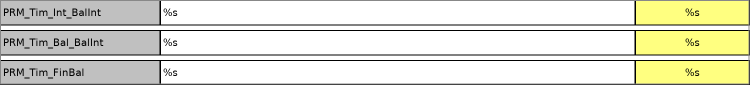
VISUALIZATION VISU_CONFIG_INTERJOINT  // 750x85
(*visualistion pour secondaire dans chambre et primaire dans sas ==> paramètres pour chambre*)
VAR_IN_OUT
	m_Input_Pompage : BLOCK_POMP_1E_PCR_PPM_ASS_ETHERCAT_SINGER;
END_VAR
    Rectangle (160,0 475x25), "%s", text list: 'TextList_Config_Pompage', text index: 17
    Rectangle (635,0 115x25), "%s", text variable: m_Input_Pompage.PRM_Tim_Int_BalInt, input disabled if: NOT Global_Variables.PRG_USER.ACTU_USER.CONF_MACHINE
        OnMouseClick: write the text variable via InputWithLimits
    Rectangle (0,0 160x25), "PRM_Tim_Int_BalInt"
    Rectangle (160,30 475x25), "%s", text list: 'TextList_Config_Pompage', text index: 18
    Rectangle (635,30 115x25), "%s", text variable: m_Input_Pompage.PRM_Tim_Bal_BalInt, input disabled if: NOT Global_Variables.PRG_USER.ACTU_USER.CONF_MACHINE
        OnMouseClick: write the text variable via InputWithLimits
    Rectangle (0,30 160x25), "PRM_Tim_Bal_BalInt"
    Rectangle (0,60 160x25), "PRM_Tim_FinBal"
    Rectangle (160,60 475x25), "%s", text list: 'TextList_Config_Pompage', text index: 19
    Rectangle (635,60 115x25), "%s", text variable: m_Input_Pompage.PRM_Tim_FinBal, input disabled if: NOT Global_Variables.PRG_USER.ACTU_USER.CONF_MACHINE
        OnMouseClick: write the text variable via InputWithLimits
END_VISUALIZATION

// ---- Visualizations/Symbole/POMPES/CRYO_CTI_V4/VISU_ETAPE_REGEN.TcVIS
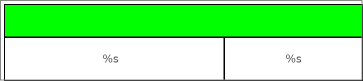
VISUALIZATION VISU_ETAPE_REGEN  // 363x81
VAR_IN_OUT
	COM: BLOCK_RS232_ONBOARD_V4;
END_VAR
    Textfield (4,37 220x44), "%s", text list: 'TextList_CryoPump', text index: COM.STEP_REGEN_ID
    Rectangle (4,4 359x33), colour toggle: COM.STATE_Regen, text list: 'TextList_CryoPump', text index: 43
    Textfield (224,37 139x44), "%s", text variable: COM.VAR_Affichage, text list: 'TextList_CryoPump', text index: COM.ID_ERREUR_REGEN
    Rectangle (4,4 359x33), colour toggle: COM.STATE_Regen, invisible if: not(COM.Regen_completed), text list: 'TextList_CryoPump', text index: 43
END_VISUALIZATION

// ---- Visualizations/Symbole/POMPES/CRYO_CTI_V4/VISU_INFO.TcVIS
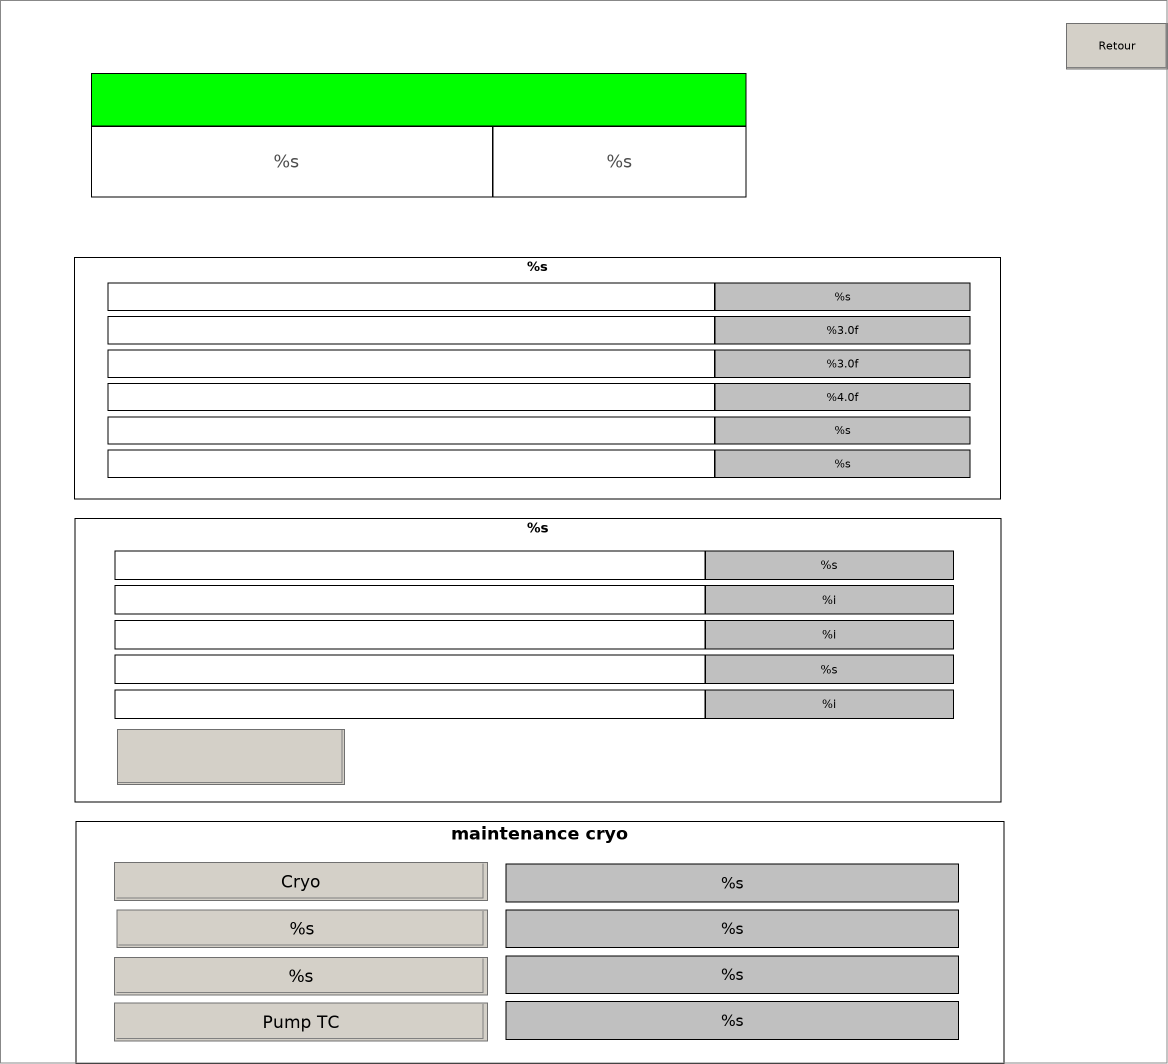
VISUALIZATION VISU_INFO  // 1168x1064
VAR_IN_OUT
	m_Input_CRYO: BLOCK_RS232_ONBOARD_V4;
	m_Input_PRG_POMPAGE: BLOCK_PRG_POMPAGE;
END_VAR
    Button (1066,23 102x46), "Retour", text list: 'GlabalTextList', text index: 16
        OnMouseClick: change screen: Previous SYN_POMPAGE
        OnMouseClick: execute { .VISU_INDEX_MANU := 0; }
    Frame (60,812 944x252), invisible if: NOT Global_Variables.PRG_USER.MANUFACTURER, input disabled if: NOT Global_Variables.PRG_USER.ACTU_USER.CONF_MACHINE OR NOT Global_Variables.PRG_USER.MANUFACTURER
        shows VISU_MAINT_CRYO_AC(COM := m_Input_CRYO)
    Frame (65,509 936x293)
        shows VISU_INFO_SUPP_POMPE(COM := m_Input_CRYO)
    Frame (68,255 933x244)
        shows VISU_RECUPERATION_ETATS(COM := m_Input_CRYO)
    Frame (84,67 662x130)
        shows VISU_ETAPE_REGEN(COM := m_Input_CRYO)
END_VISUALIZATION

// ---- Visualizations/Symbole/POMPES/CRYO_CTI_V4/VISU_INFO_SUPP_POMPE.TcVIS
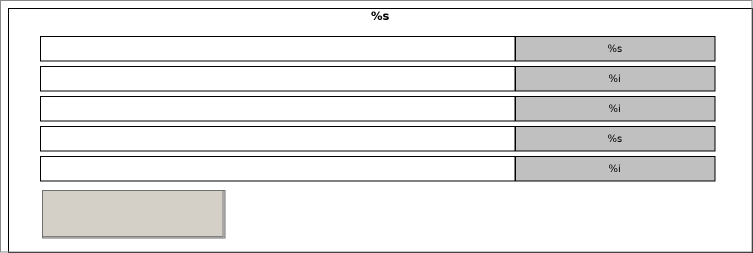
VISUALIZATION VISU_INFO_SUPP_POMPE  // 753x253
VAR_IN_OUT
	COM: BLOCK_RS232_ONBOARD_V4;
END_VAR
    RoundedRectangle (8,8 745x245), "%s", text list: 'TextList_CryoPump', text index: 87
    Rectangle (515,66 200x25), "%i", text variable: COM.Number_Of_Complete_Regen
    Rectangle (40,36 475x25), text list: 'TextList_CryoPump', text index: 47
    Rectangle (40,66 475x25), text list: 'TextList_CryoPump', text index: 48
    Rectangle (40,96 475x25), text list: 'TextList_CryoPump', text index: 49
    Rectangle (40,126 475x25), text list: 'TextList_CryoPump', text index: 50
    Rectangle (40,156 475x25), text list: 'TextList_CryoPump', text index: 51
    Rectangle (515,36 200x25), "%s", text variable: COM.Pump_Serial_Number_affiche
    Rectangle (515,96 200x25), "%i", text variable: COM.Time_Since_Last_Regen
    Rectangle (515,126 200x25), "%s", text variable: COM.SoftwareRevisionLevel
    Rectangle (515,156 200x25), "%i", text variable: COM.ElaspedTime
    Button (42,190 183x48), text list: 'TextList_CryoPump', text index: 88
        OnMouseDown: execute { COM.CO_InfoPompe:=true; }
        OnMouseUp: execute { COM.CO_InfoPompe:=false; }
END_VISUALIZATION

// ---- Visualizations/Symbole/POMPES/CRYO_CTI_V4/VISU_MAINT_CRYO_AC.TcVIS
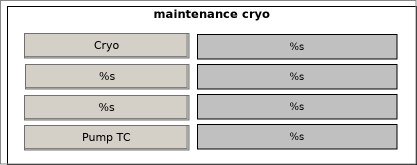
VISUALIZATION VISU_MAINT_CRYO_AC  // 417x165
VAR_IN_OUT
	COM: BLOCK_RS232_ONBOARD_V4;
END_VAR
    RoundedRectangle (7,6 410x159), "maintenance cryo", text list: 'TextList_CryoPump', text index: 97
    Rectangle (197,34 200x25), "%s", text variable: COM.PRM_PumpStartDelay, text list: 'TextList_CryoPump', text index: BOOL_TO_INT(COM.STATE_Pompe)+7
    Rectangle (197,64 200x25), "%s", text list: 'TextList_CryoPump', text index: BOOL_TO_INT(COM.STATE_Rough_valve)+37
    Rectangle (197,94 200x25), "%s", text list: 'TextList_CryoPump', text index: BOOL_TO_INT(COM.STATE_Purge_valve)+37
    Button (24,33 165x25), "Cryo"
        OnMouseClick: execute {
            IF (COM.CO_Etat=TRUE) THEN
            	com.CO_Etat:=FALSE;
            ELSE
            	com.CO_Etat:=TRUE;
            END_IF
        }
    Button (25,64 164x25), "%s", text list: 'TextList_CryoPump', text index: 41
        OnMouseClick: execute {
            IF (COM.CO_RoughValve=TRUE) THEN
            	com.CO_RoughValve:=FALSE;
            ELSE
            	com.CO_RoughValve:=TRUE;
            END_IF
        }
    Button (24,95 165x25), "%s", text list: 'TextList_CryoPump', text index: 42
        OnMouseClick: execute {
            IF (COM.CO_PurgeValve=TRUE) THEN
            	com.CO_PurgeValve:=FALSE;
            ELSE
            	com.CO_PurgeValve:=TRUE;
            END_IF
        }
    Rectangle (197,124 200x25), "%s", text list: 'TextList_CryoPump', text index: BOOL_TO_INT(COM.STATE_Pump_TC)
    Button (24,125 165x25), "Pump TC"
        OnMouseClick: execute {
            IF (COM.CO_PumpTc=TRUE) THEN
            	com.CO_PumpTc:=FALSE;
            ELSE
            	com.CO_PumpTc:=TRUE;
            END_IF
        }
END_VISUALIZATION

// ---- Visualizations/Symbole/POMPES/CRYO_CTI_V4/VISU_MESSAGE_ALERTE.TcVIS
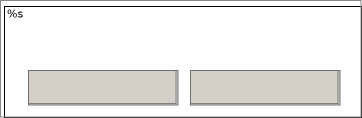
VISUALIZATION VISU_MESSAGE_ALERTE  // 362x118
VAR_IN_OUT
	COM : BLOCK_RS232_ONBOARD_V4;
	var_a_affecter: BOOL:=FALSE;
END_VAR
VAR_INPUT
	valeur_a_affecter: BOOL:=FALSE;
END_VAR
    Rectangle (4,6 358x112), "%s", text list: 'TextList_CryoPump', text index: 89
    Button (28,70 150x35), text list: 'TextList_CryoPump', text index: 92
        OnMouseClick: execute { COM.CO_Envoie_Param_Relay:=true; }
        OnMouseUp: execute { COM.CO_Envoie_Param_Relay:=false; Message_erreur_invisible:=true; }
    Button (190,70 150x35), text list: 'TextList_CryoPump', text index: 93
        OnMouseClick: execute { Message_erreur_invisible:=true; }
    Rectangle (11,30 345x30), text list: 'TextList_CryoPump', text index: 90
END_VISUALIZATION

// ---- Visualizations/Symbole/POMPES/CRYO_CTI_V4/VISU_PARAMETRAGE_RELAY.TcVIS
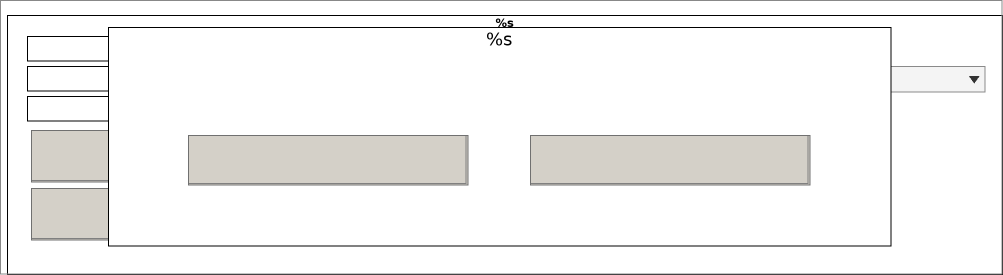
VISUALIZATION VISU_PARAMETRAGE_RELAY  // 1003x275
VAR_IN_OUT
	COM : BLOCK_RS232_ONBOARD_V4;
END_VAR
    RoundedRectangle (7,15 996x260), "%s", text list: 'TextList_CryoPump', text index: 80
    Rectangle (27,36 475x25), text list: 'TextList_CryoPump', text index: 66
    Rectangle (502,36 349x25), "%i", text variable: COM.PRM_Relay, input disabled if: NOT Global_Variables.PRG_USER.ACTU_USER.CONF_MACHINE
        OnMouseClick: write COM.PRM_Relay via Edit, min 1, max 2
    Rectangle (27,66 475x25), text list: 'TextList_CryoPump', text index: 67
    Rectangle (27,96 475x25), invisible if: COM.VAR_Visibilite_valeur_relay, text list: 'TextList_CryoPump', text index: 68
    Rectangle (502,96 349x25), "%i", text variable: COM.PRM_Valeur, invisible if: COM.VAR_Visibilite_valeur_relay, input disabled if: NOT Global_Variables.PRG_USER.ACTU_USER.CONF_MACHINE
        OnMouseClick: write COM.PRM_Valeur via Edit
    Button (31,130 244x52), input disabled if: NOT Global_Variables.PRG_USER.ACTU_USER.CONF_MACHINE, text list: 'TextList_CryoPump', text index: 69
        OnMouseDown: execute { COM.Message_alerte_invisible:=false; }
    Rectangle (485,158 200x26), text list: 'TextList_CryoPump', text index: COM.VAR_Affichage_Commande_Relay
    Rectangle (685,158 200x26), "%s", text variable: COM.VAR_Affichage_Valeur_Relay
    Rectangle (685,133 200x26), "mode", text list: 'TextList_CryoPump', text index: BOOL_TO_INT(COM.TAB_Affichage_Mode_relay[COM.PRM_Relay])+81
    Rectangle (485,184 200x26), "delay", text list: 'TextList_CryoPump', text index: 74
    Rectangle (685,184 200x26), "%s sec", text variable: COM.VAR_Affichage_ValeurTIME_Relay
    Button (31,188 244x52), input disabled if: NOT Global_Variables.PRG_USER.ACTU_USER.CONF_MACHINE, text list: 'TextList_CryoPump', text index: 85
        OnMouseDown: execute { COM.Message_alerte_invisible:=false; }
    ComboBoxInteger (503,66 482x26), variable: COM.PRM_Action, input disabled if: NOT Global_Variables.PRG_USER.ACTU_USER.CONF_MACHINE, text list: 'TextList_Cryo_Relays_Parameters'
    Button (281,130 198x52), text list: 'TextList_CryoPump', text index: 88
        OnMouseDown: execute { COM.CO_Lecture_Relay:=TRUE; }
        OnMouseUp: execute { COM.CO_Lecture_Relay:=false; }
    Button (281,188 197x52), input disabled if: NOT Global_Variables.PRG_USER.ACTU_USER.CONF_MACHINE, text list: 'TextList_CryoPump', text index: 36
        OnMouseDown: execute { COM.Message_confirm_invisible:=false; }
        OnMouseUp: execute {  }
    Group (109,27 782x218)
        Rectangle (0,0 587x176), "%s", invisible if: COM.Message_alerte_invisible, text list: 'TextList_CryoPump', text index: 89
        Rectangle (6,39 579x68), "%s", invisible if: COM.Message_alerte_invisible, text list: 'TextList_CryoPump', text index: 90
        Button (60,120 213x42), invisible if: COM.Message_alerte_invisible, text list: 'TextList_CryoPump', text index: 92
            OnMouseDown: execute { COM.CO_Envoie_Param_Relay:=true; }
            OnMouseUp: execute { COM.Message_alerte_invisible:=TRUE; }
            OnMouseUp: execute { COM.CO_Envoie_Param_Relay:=false; }
        Button (323,120 211x41), invisible if: COM.Message_alerte_invisible, text list: 'TextList_CryoPump', text index: 93
            OnMouseDown: execute { COM.Message_alerte_invisible:=true; }
    Group (109,28 782x216), invisible if: COM.Message_alerte_invisible2
        Rectangle (0,0 587x176), "%s", invisible if: COM.Message_alerte_invisible, text list: 'TextList_CryoPump', text index: 89
        Rectangle (6,39 579x68), "%s", invisible if: COM.Message_alerte_invisible, text list: 'TextList_CryoPump', text index: 90
        Button (319,120 210x40), invisible if: COM.Message_alerte_invisible, text list: 'TextList_CryoPump', text index: 93
            OnMouseDown: execute { COM.Message_alerte_invisible:=true; }
        Button (63,120 210x40), text list: 'TextList_CryoPump', text index: 85
            OnMouseDown: execute { COM.CO_Envoie_Param_Relay:=true; }
            OnMouseUp: execute { COM.CO_Envoie_Param_Relay:=FALSE; }
            OnMouseUp: execute { COM.PRM_Mode := TRUE; }
    Group (108,27 783x219)
        Rectangle (0,0 783x219), "%s", invisible if: COM.Message_confirm_invisible, text list: 'TextList_CryoPump', text index: 91
        Button (422,108 280x50), invisible if: COM.Message_confirm_invisible, text list: 'TextList_CryoPump', text index: 93
            OnMouseDown: execute { COM.Message_confirm_invisible:=true; }
        Button (80,108 280x50), invisible if: COM.Message_confirm_invisible, text list: 'TextList_CryoPump', text index: 92
            OnMouseDown: execute { COM.CO_Param_usine_Relay:=TRUE; }
            OnMouseUp: execute { COM.CO_Param_usine_Relay:=FALSE; }
            OnMouseUp: execute { COM.Message_confirm_invisible:=true; }
END_VISUALIZATION

// ---- Visualizations/Symbole/POMPES/CRYO_CTI_V4/VISU_POMPE_CRYO_CTI.TcVIS
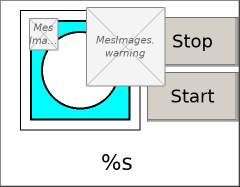
VISUALIZATION VISU_POMPE_CRYO_CTI  // 240x187
VAR_IN_OUT
	m_Input_POMPE:	BLOCK_PCR_CTI_OB;
	m_Input_COM:	BLOCK_RS232_ONBOARD_V4;
	m_Input_Forcage : BOOL;
END_VAR
    Rectangle (0,0 240x187), invisible if: TRUE
    Rectangle (30,20 100x100), colour toggle: m_Input_POMPE.STATE_Ok, invisible if: NOT m_Input_POMPE.State_on
    Rectangle (30,20 100x100), invisible if: NOT m_Input_POMPE.STATE_Ar
    Rectangle (30,20 100x100), invisible if: NOT m_Input_POMPE.STATE_Regen
    Group (41,31 78x78)
        Ellipse (0,0 78x78)
        Polyline (25,37)
        Polyline (10,4)
        Polyline (18,14)
        Polyline (26,37)
        Polyline (25,38)
    Rectangle (20,10 120x120), invisible if: NOT (m_Input_POMPE.AUTOR_On_IHM OR m_Input_POMPE.AUTOR_Off_IHM) OR NOT PRG_User.ACTU_USER.MAINTENANCE
        tap m_Input_POMPE.M_ON
    Rectangle (98,140 140x45), "%s", text variable: m_Input_POMPE.MNEMO
    Button (147,17 91x49), "Regen", invisible if: NOT m_Input_POMPE.AUTOR_Regen_IHM OR NOT PRG_User.ACTU_USER.MAINTENANCE OR m_Input_POMPE.STATE_Regen
        toggle m_Input_POMPE.M_Regen
    Button (147,17 91x49), "Stop", invisible if: NOT PRG_User.ACTU_USER.MAINTENANCE OR NOT m_Input_POMPE.STATE_Regen
        OnMouseDown: execute { m_Input_COM.CO_StopRegen:=TRUE; }
        OnMouseUp: execute { m_Input_COM.CO_StopRegen:=FALSE; }
    Button (147,72 91x49), "Start", invisible if: NOT PRG_User.ACTU_USER.MAINTENANCE OR NOT m_Input_POMPE.OUT_On OR ( NOT m_Input_COM.STATE_Pompe = 0) OR m_Input_POMPE.STATE_Regen
        OnMouseDown: execute { m_Input_Forcage:=TRUE; }
        OnMouseUp: execute { m_Input_Forcage:=FALSE; }
    Image (86,7 79x79), invisible if: NOT m_Input_POMPE.STATE_NOK, image: MesImages.warning
    Image (29,18 29x32), invisible if: NOT m_Input_COM.STATE_Pompe, image: MesImages.Flocon
END_VISUALIZATION

// ---- Visualizations/Symbole/POMPES/CRYO_CTI_V4/VISU_RECUPERATION_ETATS.TcVIS
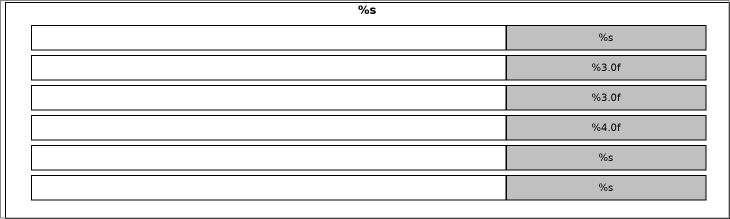
VISUALIZATION VISU_RECUPERATION_ETATS  // 730x219
VAR_IN_OUT
	COM: BLOCK_RS232_ONBOARD_V4;
END_VAR
    RoundedRectangle (5,2 725x217), "%s", text list: 'TextList_CryoPump', text index: 94
    Rectangle (506,55 200x25), "%3.0f", text variable: COM.STATE_Temperature[0]
    Rectangle (31,25 475x25), text list: 'TextList_CryoPump', text index: 4
    Rectangle (31,55 475x25), text list: 'TextList_CryoPump', text index: 5
    Rectangle (31,85 475x25), text list: 'TextList_CryoPump', text index: 6
    Rectangle (31,115 475x25), text list: 'TextList_CryoPump', text index: 53
    Rectangle (31,145 475x25), text list: 'TextList_CryoPump', text index: 39
    Rectangle (31,175 475x25), text list: 'TextList_CryoPump', text index: 40
    Rectangle (506,25 200x25), "%s", text variable: COM.PRM_PumpStartDelay, text list: 'TextList_CryoPump', text index: BOOL_TO_INT(COM.STATE_Pompe)+7
    Rectangle (506,85 200x25), "%3.0f", text variable: COM.STATE_Temperature[1]
    Rectangle (506,115 200x25), "%4.0f", text variable: COM.STATE_Pressure
    Rectangle (506,145 200x25), "%s", text list: 'TextList_CryoPump', text index: BOOL_TO_INT(COM.STATE_Rough_valve)+37
    Rectangle (506,175 200x25), "%s", text list: 'TextList_CryoPump', text index: BOOL_TO_INT(COM.STATE_Purge_valve)+37
END_VISUALIZATION

// ---- Visualizations/Symbole/POMPES/CRYO_CTI_V4/VISU_REGENERATION.TcVIS
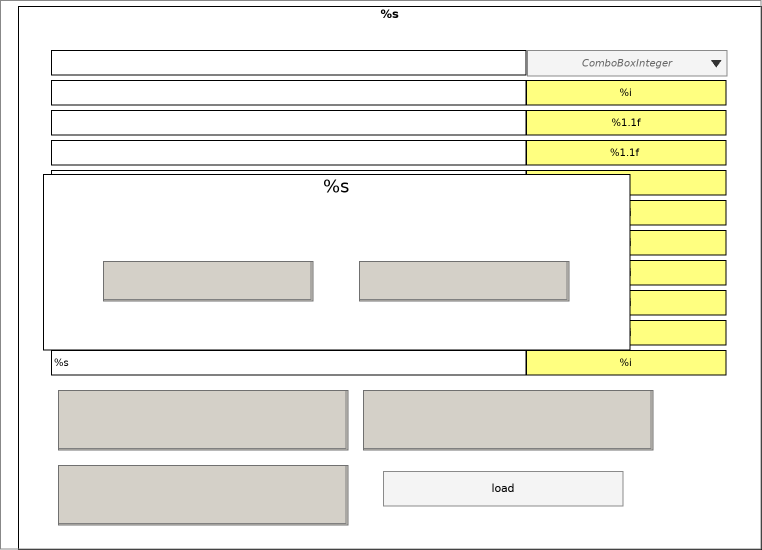
VISUALIZATION VISU_REGENERATION  // 762x550
VAR_IN_OUT
	COM: BLOCK_RS232_ONBOARD_V4;
END_VAR
    RoundedRectangle (18,6 744x544), "%s", text list: 'TextList_CryoPump', text index: 98
    Rectangle (51,50 475x25), text list: 'TextList_CryoPump', text index: 45
    Rectangle (526,140 200x25), "%1.1f", text variable: COM.PRM_PumpRestartDelay, input disabled if: NOT Global_Variables.PRG_USER.ACTU_USER.CONF_MACHINE
        OnMouseClick: write COM.PRM_PumpRestartDelay via Edit
    Rectangle (51,110 475x25), text list: 'TextList_CryoPump', text index: 57
    Rectangle (51,140 475x25), text list: 'TextList_CryoPump', text index: 11
    Rectangle (51,170 475x25), text list: 'TextList_CryoPump', text index: 10
    Rectangle (51,200 475x25), text list: 'TextList_CryoPump', text index: 12
    Rectangle (51,230 475x25), text list: 'TextList_CryoPump', text index: 13
    Rectangle (51,260 475x25), text list: 'TextList_CryoPump', text index: 30
    Progressbar (383,471 240x35), "load", variable: COM.iCounter_Regen_lecture, invisible if: not(COM.VAR_Mem_CO_Lecture)
    Rectangle (526,110 200x25), "%1.1f", text variable: COM.PRM_PumpStartDelay, input disabled if: NOT Global_Variables.PRG_USER.ACTU_USER.CONF_MACHINE
        OnMouseClick: write COM.PRM_PumpStartDelay via Edit
    ComboBoxInteger (527,50 200x26), variable: COM.ID_COMBOBOX, input disabled if: NOT Global_Variables.PRG_USER.ACTU_USER.CONF_MACHINE, text list: 'TextList_CryoPump'
    Rectangle (526,170 200x25), "%i", text variable: COM.PRM_ExtendedPurgeTime, input disabled if: NOT Global_Variables.PRG_USER.ACTU_USER.CONF_MACHINE
        OnMouseClick: write COM.PRM_ExtendedPurgeTime via Edit
    Rectangle (526,200 200x25), "%i", text variable: COM.PRM_RepurgeCycles, input disabled if: NOT Global_Variables.PRG_USER.ACTU_USER.CONF_MACHINE
        OnMouseClick: write COM.PRM_RepurgeCycles via Edit
    Rectangle (526,230 200x25), "%i", text variable: COM.PRM_RepurgeTime, input disabled if: NOT Global_Variables.PRG_USER.ACTU_USER.CONF_MACHINE
        OnMouseClick: write COM.PRM_RepurgeTime via Edit
    Rectangle (526,260 200x25), "%i", text variable: COM.PRM_ROR, input disabled if: NOT Global_Variables.PRG_USER.ACTU_USER.CONF_MACHINE
        OnMouseClick: write COM.PRM_ROR via Edit
    Rectangle (51,290 475x25), text list: 'TextList_CryoPump', text index: 14
    Rectangle (526,290 200x25), "%i", text variable: COM.PRM_RORCycles, input disabled if: NOT Global_Variables.PRG_USER.ACTU_USER.CONF_MACHINE
        OnMouseClick: write COM.PRM_RORCycles via Edit
    Rectangle (51,320 475x25), text list: 'TextList_CryoPump', text index: 29
    Rectangle (526,320 200x25), "%i", text variable: COM.PRM_RoughToPressure, input disabled if: NOT Global_Variables.PRG_USER.ACTU_USER.CONF_MACHINE
        OnMouseClick: write COM.PRM_RoughToPressure via Edit
    Rectangle (51,80 475x25), text list: 'TextList_CryoPump', text index: 17
    Rectangle (526,80 200x25), "%i", text variable: COM.PRM_StartUpTemperature, input disabled if: NOT Global_Variables.PRG_USER.ACTU_USER.CONF_MACHINE
        OnMouseClick: write COM.PRM_StartUpTemperature via Edit
    Progressbar (383,471 240x35), "load", variable: COM.iCounter_Regen_ecriture, invisible if: not(COM.VAR_Mem_CO_Ecriture)
    Button (58,390 290x60), text list: 'TextList_CryoPump', text index: 18
        OnMouseDown: toggle COM.CO_Lecture
    Button (363,390 290x60), input disabled if: NOT Global_Variables.PRG_USER.ACTU_USER.CONF_MACHINE, text list: 'TextList_CryoPump', text index: 19
        OnMouseDown: toggle COM.CO_Ecriture
        OnMouseUp: execute { COM.CO_Ecriture:= false; }
    Button (58,465 290x60), input disabled if: NOT Global_Variables.PRG_USER.ACTU_USER.CONF_MACHINE, text list: 'TextList_CryoPump', text index: 36
        OnMouseDown: execute { COM.Message_confirm_invisible_regen:=false; }
    Rectangle (51,350 475x25), "%s", text list: 'TextList_CryoPump', text index: 96
    Rectangle (526,350 200x25), "%i", text variable: COM.PRM_1st_stage_control_temp, input disabled if: NOT Global_Variables.PRG_USER.ACTU_USER.CONF_MACHINE OR NOT Global_Variables.PRG_USER.MANUFACTURER
        OnMouseClick: write COM.PRM_1st_stage_control_temp via Edit
    Group (43,174 692x182), invisible if: COM.Message_confirm_invisible_regen
        Rectangle (0,0 587x176), "%s", text list: 'TextList_CryoPump', text index: 91
        Button (316,87 210x40), text list: 'TextList_CryoPump', text index: 93
            OnMouseDown: execute { COM.Message_confirm_invisible_regen:=true; }
        Button (60,87 210x40), text list: 'TextList_CryoPump', text index: 92
            OnMouseDown: execute { COM.CO_Param_ParDefaut:=TRUE; }
            OnMouseUp: execute { COM.CO_Param_ParDefaut:= false; }
            OnMouseUp: execute { COM.Message_confirm_invisible_regen:=true; }
END_VISUALIZATION

// ---- Visualizations/Symbole/POMPES/CRYO_CTI_V4/VISU_TEMP_POMP_CRYO_SOLO.TcVIS
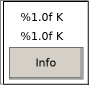
VISUALIZATION VISU_TEMP_POMP_CRYO_SOLO  // 89x85
VAR_IN_OUT
	m_Input_CRYO: BLOCK_RS232_ONBOARD_V4;
	m_Input_PRG_POMPAGE: BLOCK_PRG_POMPAGE;
END_VAR
VAR_INPUT
	m_Input_NumFrame_Manu:	USINT;		(*numéro de frame à afficher dans le synoptique MANUEL*)
	m_Input_INDEX_CRYO : INT;
END_VAR
    RoundedRectangle (3,1 86x84)
    Rectangle (7,8 70x19), "%1.0f K", text variable: PRG_POMPAGE.COM_CRYOS.STATE_Temperature[0]
    Rectangle (7,27 70x19), "%1.0f K", text variable: PRG_POMPAGE.COM_CRYOS.STATE_Temperature[1]
    Button (9,47 74x32), "Info"
        OnMouseClick: change screen: SYN_MANUEL
        OnMouseClick: execute { .VISU_INDEX_MANU := m_Input_NumFrame_Manu; }
END_VISUALIZATION

// ---- Visualizations/Symbole/POMPES/VISU_POMPE_PRIMAIRE.TcVIS
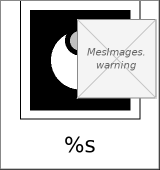
VISUALIZATION VISU_POMPE_PRIMAIRE  // 160x170
VAR_IN_OUT
	m_Input_POMPE : BLOCK_PPM;
END_VAR
    Rectangle (0,0 160x170), invisible if: TRUE
    Rectangle (10,130 140x30), "%s", text variable: m_Input_POMPE.MNEMO
    Rectangle (30,10 100x100)
    Rectangle (30,10 100x100), colour toggle: (m_Input_POMPE.STATE_ON) <> 0, invisible if: NOT m_Input_POMPE.STATE_ON AND NOT m_Input_POMPE.STATE_OFF
    Group (46,26 68x68)
        Ellipse (0,0 68x68)
        Ellipse (19,0 29x29)
    Rectangle (20,0 120x119), invisible if: NOT (m_Input_POMPE.Autor_ON_IHM OR m_Input_POMPE.Autor_OFF_IHM) OR NOT PRG_User.ACTU_USER.MAINTENANCE
        tap m_Input_POMPE.M_ON
    Image (77,19 79x79), invisible if: NOT m_Input_POMPE.STATE_NOK, image: MesImages.warning
END_VISUALIZATION

// ---- Visualizations/Symbole/POMPES/VISU_POMPE_PRIMAIRE_DEF.TcVIS
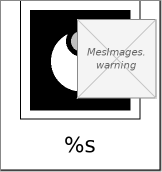
VISUALIZATION VISU_POMPE_PRIMAIRE_DEF  // 162x172
VAR_IN_OUT
	m_Input_POMPE : BLOCK_PPM_DEF;
END_VAR
    Rectangle (0,0 160x170), invisible if: TRUE
    Rectangle (10,130 140x30), "%s", text variable: m_Input_POMPE.MNEMO
    Rectangle (30,10 100x100)
    Rectangle (30,10 100x100), colour toggle: (m_Input_POMPE.STATE_ON) <> 0, invisible if: NOT m_Input_POMPE.STATE_ON AND NOT m_Input_POMPE.STATE_OFF
    Group (46,26 68x68)
        Ellipse (0,0 70x70)
        Ellipse (20,0 30x30)
    Rectangle (20,0 120x119), invisible if: NOT (m_Input_POMPE.Autor_ON_IHM OR m_Input_POMPE.Autor_OFF_IHM) OR NOT PRG_User.ACTU_USER.MAINTENANCE
        tap m_Input_POMPE.M_ON
    Image (77,19 79x79), invisible if: NOT m_Input_POMPE.STATE_NOK, image: MesImages.warning
END_VISUALIZATION

// ---- Visualizations/Symbole/POMPES/VISU_POMPE_ROOTS.TcVIS
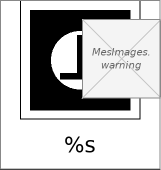
VISUALIZATION VISU_POMPE_ROOTS  // 161x170
VAR_IN_OUT
	m_Input_POMPE : BLOCK_PPM;
END_VAR
    Rectangle (0,0 160x170), invisible if: TRUE
    Rectangle (10,130 140x30), "%s", text variable: m_Input_POMPE.MNEMO
    Rectangle (30,10 100x100)
    Rectangle (30,10 100x100), colour toggle: (m_Input_POMPE.STATE_ON) <> 0, invisible if: NOT m_Input_POMPE.STATE_ON AND NOT m_Input_POMPE.STATE_OFF
    Ellipse (46,26 68x68)
    Rectangle (20,0 120x119), invisible if: NOT (m_Input_POMPE.Autor_ON_IHM OR m_Input_POMPE.Autor_OFF_IHM) OR NOT PRG_User.ACTU_USER.MAINTENANCE
        tap m_Input_POMPE.M_ON
    Rectangle (77,35 6x39)
    Rectangle (60,73 41x6)
    Image (82,19 79x79), invisible if: NOT m_Input_POMPE.STATE_NOK, image: MesImages.warning
END_VISUALIZATION

// ---- Visualizations/Symbole/POMPES/VISU_POMPE_TURBO.TcVIS
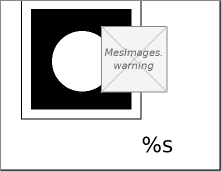
VISUALIZATION VISU_POMPE_TURBO  // 222x172
VAR_IN_OUT
	m_Input_POMPE : BLOCK_PPM_DEF;
END_VAR
    Rectangle (0,0 220x170), invisible if: TRUE
    Rectangle (96,130 123x30), "%s", text variable: m_Input_POMPE.MNEMO
    Rectangle (31,9 100x100), colour toggle: (m_Input_POMPE.OUT_ON) <> 0
    Rectangle (31,9 100x100), colour toggle: (m_Input_POMPE.STATE_ON) <> 0, invisible if: NOT m_Input_POMPE.STATE_ON AND NOT m_Input_POMPE.STATE_OFF
    Group (47,26 68x68)
        Ellipse (0,0 70x70)
        Polyline (65,36)
        Polyline (5,42)
        Polyline (15,42)
        Polyline (25,42)
        Polyline (35,42)
        Polyline (45,42)
        Polyline (55,42)
        Polyline (65,42)
    Rectangle (21,0 120x119), invisible if: NOT (m_Input_POMPE.Autor_ON_IHM OR m_Input_POMPE.Autor_OFF_IHM) OR NOT PRG_User.ACTU_USER.MAINTENANCE
        tap m_Input_POMPE.M_ON
    Image (101,26 66x66), invisible if: NOT m_Input_POMPE.STATE_NOK, image: MesImages.warning
END_VISUALIZATION

// ---- Visualizations/Symbole/POMPES/VISU_POMPE_TURBO_VPURGE.TcVIS
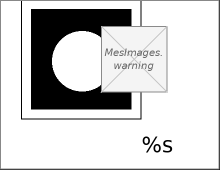
VISUALIZATION VISU_POMPE_TURBO_VPURGE  // 220x170
VAR_IN_OUT
	m_Input_POMPE : BLOCK_PPM_DEF_VPURGE;
END_VAR
    Rectangle (0,0 220x170), invisible if: TRUE
    Rectangle (96,130 123x30), "%s", text variable: m_Input_POMPE.MNEMO
    Rectangle (31,9 100x100), colour toggle: (m_Input_POMPE.OUT_ON) <> 0
    Rectangle (31,9 100x100), colour toggle: (m_Input_POMPE.STATE_ON) <> 0, invisible if: NOT m_Input_POMPE.STATE_ON AND NOT m_Input_POMPE.STATE_OFF
    Group (47,26 68x68)
        Ellipse (0,0 70x70)
        Polyline (65,36)
        Polyline (5,42)
        Polyline (15,42)
        Polyline (25,42)
        Polyline (35,42)
        Polyline (45,42)
        Polyline (55,42)
        Polyline (65,42)
    Rectangle (21,0 120x119), invisible if: NOT (m_Input_POMPE.Autor_ON_IHM OR m_Input_POMPE.Autor_OFF_IHM) OR NOT PRG_User.ACTU_USER.MAINTENANCE
        tap m_Input_POMPE.M_ON
    Image (101,26 66x66), invisible if: NOT m_Input_POMPE.STATE_NOK, image: MesImages.warning
END_VISUALIZATION

// ---- Visualizations/Symbole/PROCEDE/VISU_INFO_PROCESS.TcVIS
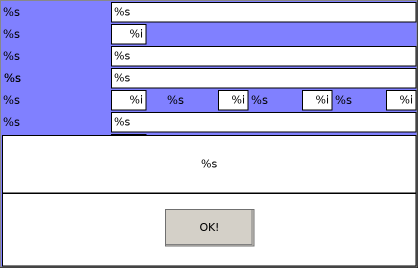
VISUALIZATION VISU_INFO_PROCESS  // 418x268
    Rectangle (0,0 418x268)
    Button (296,202 120x30), "%s", input disabled if: NOT (PRG_USER.ACTU_USER.PRODUCTION), text list: 'TextList_Process', text index: 26
        toggle EXECPROC.M_LOAD_PROCESS
    Rectangle (0,2 110x20), "%s", text list: 'TextList_Process', text index: 7
    Rectangle (111,2 305x20), "%s", text variable: EXECPROC.PRM_PROCESS
    Rectangle (0,24 110x20), "%s", text list: 'TextList_Process', text index: 8
    Rectangle (111,24 35x20), "%i", text variable: EXECPROC.STATE_STEP
    Rectangle (0,46 110x20), "%s", text list: 'TextList_Process', text index: 9
    Rectangle (111,46 305x20), "%s", text list: 'TextList_Type_Etape', text index: EXECPROC.PRM_TYPE_ETAPE
    Rectangle (0,90 110x20), "%s", invisible if: MAIN.STEP_EMPILEMENT.OP_RUN.AR, text list: 'TextList_Process', text index: 11
    Rectangle (111,90 35x20), "%i", text variable: MAIN.STEP_EMPILEMENT.STATE_LAYER, invisible if: MAIN.STEP_EMPILEMENT.OP_RUN.AR
    Rectangle (0,112 110x20), "%s", invisible if: MAIN.STEP_EMPILEMENT.OP_RUN.AR, text list: 'TextList_Process', text index: 12
    Rectangle (111,112 305x20), "%s", text variable: MAIN.STEP_EMPILEMENT.STATE_LAYER_TEXT, invisible if: MAIN.STEP_EMPILEMENT.OP_RUN.AR
    Rectangle (164,90 55x20), "%s", invisible if: MAIN.STEP_EMPILEMENT.OP_RUN.AR OR (MAIN.STEP_EMPILEMENT.PRM_NB_LOOP = 0), text list: 'TextList_Process', text index: 13
    Rectangle (248,90 55x20), "%s", invisible if: MAIN.STEP_EMPILEMENT.OP_RUN.AR OR (MAIN.STEP_EMPILEMENT.PRM_NB_LOOP = 0), text list: 'TextList_Process', text index: 14
    Rectangle (218,90 30x20), "%i", text variable: MAIN.STEP_EMPILEMENT.PRM_NB_LOOP, invisible if: MAIN.STEP_EMPILEMENT.OP_RUN.AR OR (MAIN.STEP_EMPILEMENT.PRM_NB_LOOP = 0)
    Rectangle (302,90 30x20), "%i", text variable: MAIN.STEP_EMPILEMENT.PRM_LOOP_FIRST_LAYER, invisible if: MAIN.STEP_EMPILEMENT.OP_RUN.AR OR (MAIN.STEP_EMPILEMENT.PRM_NB_LOOP = 0)
    Rectangle (332,90 55x20), "%s", invisible if: MAIN.STEP_EMPILEMENT.OP_RUN.AR OR (MAIN.STEP_EMPILEMENT.PRM_NB_LOOP = 0), text list: 'TextList_Process', text index: 15
    Rectangle (386,90 30x20), "%i", text variable: MAIN.STEP_EMPILEMENT.PRM_LOOP_LAST_LAYER, invisible if: MAIN.STEP_EMPILEMENT.OP_RUN.AR OR (MAIN.STEP_EMPILEMENT.PRM_NB_LOOP = 0)
    Rectangle (0,134 110x20), "%s", invisible if: PRG_EVAP.EVAPS1.OP_Marche.AR, text list: 'TextList_Process', text index: 16
    Rectangle (0,156 110x20), "%s", invisible if: PRG_EVAP.EVAPS1.OP_Marche.AR, text list: 'TextList_Process', text index: 17
    Rectangle (0,178 110x20), "%s", invisible if: PRG_EVAP.EVAPS1.OP_Marche.AR, text list: 'TextList_Process', text index: 18
    Rectangle (111,134 35x20), "%i", text variable: PRG_EVAP.EVAPS1.STATE_Segment, invisible if: PRG_EVAP.EVAPS1.OP_Marche.AR
    Rectangle (111,156 305x20), "%s", text variable: PRG_EVAP.EVAPS1.STATE_Temps_segment, invisible if: PRG_EVAP.EVAPS1.OP_Marche.AR
    Rectangle (111,178 305x20), "%s", text variable: PRG_EVAP.EVAPS1.TIMER_Temps_Couche.ET, invisible if: PRG_EVAP.EVAPS1.OP_Marche.AR, text index: 18
    Button (149,202 120x30), "%s", input disabled if: NOT (PRG_USER.ACTU_USER.PRODUCTION AND MAIN.STEP_EMPILEMENT.AUTOR_NEXT_LAYER), text list: 'TextList_Process', text index: 19
        toggle MAIN.STEP_EMPILEMENT.M_NEXT_LAYER
    Button (2,234 120x30), "%s", input disabled if: NOT (PRG_USER.ACTU_USER.PRODUCTION AND MACHINE.AUTOR_Inter_Prod_ihm), text list: 'TextList_Process', text index: 20
        toggle MACHINE.M_inter_Prod
    Button (149,234 120x30), "%s", input disabled if: NOT (PRG_USER.ACTU_USER.PRODUCTION AND MACHINE.AUTOR_Repris_Prod_ihm), text list: 'TextList_Process', text index: 21
        toggle MACHINE.M_Reprise_Prod
    Button (296,234 120x30), "%s", input disabled if: NOT (PRG_USER.ACTU_USER.PRODUCTION AND MACHINE.AUTOR_Stop_Prod_Ihm), text list: 'TextList_Process', text index: 22
        toggle MACHINE.M_Stop_Prod
    Button (2,202 120x30), "%s", input disabled if: NOT (PRG_USER.ACTU_USER.PRODUCTION AND EXECPROC.AUTOR_NEXT_STEP), text list: 'TextList_Process', text index: 23
        toggle EXECPROC.M_NEXT_STEP
    Rectangle (111,68 305x20), "/", invisible if: NOT MAIN.STEP_TIMER.I_ON
    Rectangle (126,69 121x18), "%s", text variable: MAIN.STEP_TIMER.TIMER.ET, invisible if: NOT MAIN.STEP_TIMER.I_ON
    Rectangle (288,69 121x18), "%s", text variable: MAIN.STEP_TIMER.TIMER.PT, invisible if: NOT MAIN.STEP_TIMER.I_ON
    Rectangle (1,68 110x20), "%s", invisible if: NOT EXECPROC.RQ_EXEC_STEP[1], text list: 'TextList_Process', text index: 12
    Rectangle (111,68 305x20), "%s", text variable: PRG_POMPAGE.PRM_Pr_Pumping_OK, invisible if: NOT EXECPROC.RQ_EXEC_STEP[1]
    Rectangle (0,179 110x20), "%s", invisible if: PRG_EVAP.EVAPS2.OP_Marche.AR, text list: 'TextList_Process', text index: 18
    Rectangle (0,135 110x20), "%s", invisible if: PRG_EVAP.EVAPS2.OP_Marche.AR, text list: 'TextList_Process', text index: 16
    Rectangle (0,157 110x20), "%s", invisible if: PRG_EVAP.EVAPS2.OP_Marche.AR, text list: 'TextList_Process', text index: 17
    Rectangle (111,135 35x20), "%i", text variable: PRG_EVAP.EVAPS2.STATE_Segment, invisible if: PRG_EVAP.EVAPS2.OP_Marche.AR
    Rectangle (111,157 305x20), "%s", text variable: PRG_EVAP.EVAPS2.STATE_Temps_segment, invisible if: PRG_EVAP.EVAPS2.OP_Marche.AR
    Rectangle (111,179 305x20), "%s", text variable: PRG_EVAP.EVAPS2.TIMER_Temps_Couche.ET, invisible if: PRG_EVAP.EVAPS2.OP_Marche.AR, text index: 18
    Rectangle (0,178 110x20), "%s", invisible if: PRG_EVAP.EVAPS3.OP_Marche.AR, text list: 'TextList_Process', text index: 18
    Rectangle (0,134 110x20), "%s", invisible if: PRG_EVAP.EVAPS3.OP_Marche.AR, text list: 'TextList_Process', text index: 16
    Rectangle (0,156 110x20), "%s", invisible if: PRG_EVAP.EVAPS3.OP_Marche.AR, text list: 'TextList_Process', text index: 17
    Rectangle (111,134 35x20), "%i", text variable: PRG_EVAP.EVAPS3.STATE_Segment, invisible if: PRG_EVAP.EVAPS3.OP_Marche.AR
    Rectangle (111,156 305x20), "%s", text variable: PRG_EVAP.EVAPS3.STATE_Temps_segment, invisible if: PRG_EVAP.EVAPS3.OP_Marche.AR
    Rectangle (111,178 305x20), "%s", text variable: PRG_EVAP.EVAPS3.TIMER_Temps_Couche.ET, invisible if: PRG_EVAP.EVAPS3.OP_Marche.AR, text index: 18
    Rectangle (2,193 414x73), invisible if: NOT MAIN.STEP_USER_ACK.STATE_EC
    Button (165,209 89x37), "OK!", invisible if: NOT MAIN.STEP_USER_ACK.STATE_EC
        tap MAIN.STEP_USER_ACK.M_GOON
    Rectangle (2,135 414x58), "%s", text variable: MAIN.STEP_USER_ACK.PRM_TEXT, invisible if: NOT MAIN.STEP_USER_ACK.STATE_EC
    Rectangle (1,68 110x20), "%s", invisible if: MAIN.STEP_EFFLUVAGE.OP_RUN.AR or true, text list: 'TextList_Process', text index: 10
END_VISUALIZATION

// ---- Visualizations/Symbole/PROCEDE/VISU_MODE_QUARTZ.TcVIS
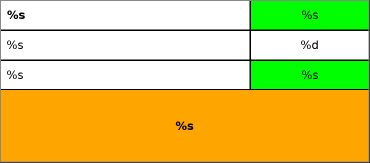
VISUALIZATION VISU_MODE_QUARTZ  // 370x163
VAR_INPUT
	m_input_Mode_Quartz:		BLOCK_1RUN_1QUARTZ;
END_VAR
    Rectangle (0,0 250x30), "%s", text list: 'TextList_1Run_1Quartz', text index: 0
    Rectangle (0,30 250x30), "%s", invisible if: not m_input_Mode_Quartz.STATE_Mode, text list: 'TextList_1Run_1Quartz', text index: 4
    Rectangle (0,60 250x30), "%s", text list: 'TextList_1Run_1Quartz', text index: 3
    Rectangle (250,0 120x30), "%s", colour toggle: MACHINE.CONF_Standby_Auto, invisible if: m_input_Mode_Quartz.STATE_Mode, text list: 'TextList_1Run_1Quartz', text index: 2
    Rectangle (250,0 120x30), "%s", colour toggle: MACHINE.CONF_Standby_Auto, invisible if: not m_input_Mode_Quartz.STATE_Mode, text list: 'TextList_1Run_1Quartz', text index: 1
    Rectangle (250,60 120x30), "%s", colour toggle: MACHINE.CONF_Standby_Auto, invisible if: m_input_Mode_Quartz.STATE_RAZ_Quartz, text list: 'TextList_1Run_1Quartz', text index: 2
    Rectangle (250,60 120x30), "%s", colour toggle: MACHINE.CONF_Standby_Auto, invisible if: not m_input_Mode_Quartz.STATE_RAZ_Quartz, text list: 'TextList_1Run_1Quartz', text index: 1
    Rectangle (250,30 120x30), "%d", text variable: m_input_Mode_Quartz.STATE_Next_Quartz, invisible if: not m_input_Mode_Quartz.STATE_Mode
    Rectangle (0,89 370x74), "%s", invisible if: not m_input_Mode_Quartz.RQ_Disp_Change_Quartz, text list: 'TextList_1Run_1Quartz', text index: 5
    Rectangle (250,0 120x30), colour toggle: MACHINE.CONF_Standby_Auto, invisible if: MODE_QUARTZ_PROD.I_Prod
        tap MODE_QUARTZ_PROD.M_Mode
    Rectangle (250,59 120x30), colour toggle: MACHINE.CONF_Standby_Auto, invisible if: not MODE_QUARTZ_PROD.STATE_Mode
        tap MODE_QUARTZ_PROD.M_RAZ_Quartz
END_VISUALIZATION

// ---- Visualizations/Symbole/PS/VISU_PS.TcVIS
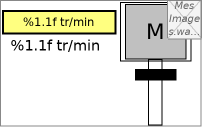
VISUALIZATION VISU_PS  // 202x127
VAR_IN_OUT
	m_Input_MOTOR : BLOCK_VARIATEUR_MOTEUR;
END_VAR
    Rectangle (148,59 14x66)
    RoundedRectangle (125,4 61x55), "M", colour toggle: (m_Input_MOTOR.STATE_On) <> 0
    Rectangle (3,34 112x23), "%1.1f tr/min", text variable: m_Input_MOTOR.STATE_Consigne, invisible if: TRUE
    RoundedRectangle (2,10 114x24), "%1.1f tr/min", text variable: m_Input_MOTOR.PRM_Cons_Vitesse, input disabled if: NOT Global_Variables.PRG_USER.ACTU_USER.MAINTENANCE OR NOT m_Input_MOTOR.Manual
        OnMouseDown: write the text variable via InputWithLimits, min 0.2, max 20.0
    Rectangle (135,69 41x11)
    Rectangle (120,2 71x59), invisible if: NOT (m_Input_MOTOR.Autor_OFF_IHM) OR NOT PRG_User.ACTU_USER.MAINTENANCE
        tap m_Input_MOTOR.M_OFF
    Rectangle (120,2 71x59), invisible if: NOT (m_Input_MOTOR.Autor_ON_IHM) OR NOT PRG_User.ACTU_USER.MAINTENANCE
        tap m_Input_MOTOR.M_ON
    Image (167,-2 35x41), invisible if: NOT m_Input_MOTOR.STATE_NOK, image: MesImages.warning
END_VISUALIZATION

// ---- Visualizations/Symbole/SERVITUDES/VISU_CONF_LIGNE_EAU_FLOWTEMP.TcVIS
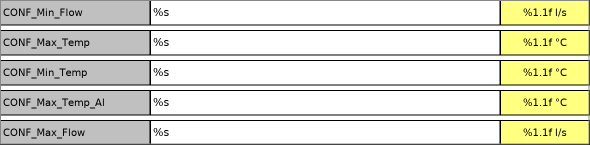
VISUALIZATION VISU_CONF_LIGNE_EAU_FLOWTEMP  // 590x145
VAR_IN_OUT
	m_Input_LIGNE_CONF_EAU : BLOCK_LIGNE_REF_FLOWTEMP;
END_VAR
    Rectangle (0,0 150x25), "CONF_Min_Flow"
    Rectangle (0,120 150x25), "CONF_Max_Flow", invisible if: true
    Rectangle (0,60 150x25), "CONF_Min_Temp"
    Rectangle (0,30 150x25), "CONF_Max_Temp"
    Rectangle (0,90 150x25), "CONF_Max_Temp_Al"
    Rectangle (500,0 90x25), "%1.1f l/s", text variable: m_Input_LIGNE_CONF_EAU.CONF_Min_Flow, input disabled if: NOT Global_Variables.PRG_USER.ACTU_USER.CONF_MACHINE OR m_Input_LIGNE_CONF_EAU.CONF_Max_Flow <= 0
        OnMouseClick: write the text variable via VisuDialogs.NumpadExtended, min 0, max m_Input_LIGNE_CONF_EAU.CONF_Max_Flow
    Rectangle (500,120 90x25), "%1.1f l/s", text variable: m_Input_LIGNE_CONF_EAU.CONF_Max_Flow, invisible if: true, input disabled if: NOT Global_Variables.PRG_USER.ACTU_USER.CONF_MACHINE
        OnMouseClick: write the text variable via VisuDialogs.NumpadExtended, min m_Input_LIGNE_CONF_EAU.CONF_Min_Flow, max 100
    Rectangle (500,60 90x25), "%1.1f °C", text variable: m_Input_LIGNE_CONF_EAU.CONF_Min_Temp, input disabled if: NOT Global_Variables.PRG_USER.ACTU_USER.CONF_MACHINE OR m_Input_LIGNE_CONF_EAU.CONF_Max_Temp <= 0
        OnMouseClick: write the text variable via VisuDialogs.NumpadExtended, min 0, max m_Input_LIGNE_CONF_EAU.CONF_Max_Temp
    Rectangle (500,30 90x25), "%1.1f °C", text variable: m_Input_LIGNE_CONF_EAU.CONF_Max_Temp, input disabled if: NOT Global_Variables.PRG_USER.ACTU_USER.CONF_MACHINE
        OnMouseClick: write the text variable via VisuDialogs.NumpadExtended, min m_Input_LIGNE_CONF_EAU.CONF_Min_Temp, max 100
    Rectangle (500,90 90x25), "%1.1f °C", text variable: m_Input_LIGNE_CONF_EAU.CONF_Max_Temp_AL, input disabled if: NOT Global_Variables.PRG_USER.ACTU_USER.CONF_MACHINE OR m_Input_LIGNE_CONF_EAU.CONF_Max_Temp <= 0
        OnMouseClick: write the text variable via VisuDialogs.NumpadExtended, min 0, max m_Input_LIGNE_CONF_EAU.CONF_Max_Temp
    Rectangle (150,0 350x25), "%s", text list: 'TextList_Servitudes', text index: 1
    Rectangle (150,120 350x25), "%s", invisible if: true, text list: 'TextList_Servitudes', text index: 2
    Rectangle (150,60 350x25), "%s", text list: 'TextList_Servitudes', text index: 3
    Rectangle (150,30 350x25), "%s", text list: 'TextList_Servitudes', text index: 4
    Rectangle (150,90 350x25), "%s", text list: 'TextList_Servitudes', text index: 5
END_VISUALIZATION

// ---- Visualizations/Symbole/SERVITUDES/VISU_LIGNE_EAU.TcVIS
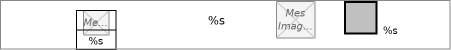
VISUALIZATION VISU_LIGNE_EAU  // 451x50
VAR_IN_OUT
	m_Input_LIGNE_EAU : BLOCK_LIGNE_REF;
END_VAR
    Polyline (451,20)
    Polyline (80,20)
    Polyline (129,20)
    Polygon (140,20)
    Polygon (317,20)
    Rectangle (380,15 65x31), "%s", text variable: m_Input_LIGNE_EAU.mnemo_DEX, invisible if: m_Input_LIGNE_EAU.CONF_NO_DexT
    Group (344,1 33x33), invisible if: (m_Input_LIGNE_EAU.CONF_NO_DexT) <> 0
        Rectangle (0,0 33x33), colour toggle: (m_Input_LIGNE_EAU.IN_DExT) <> 0
        Polyline (16,8)
        Polyline (24,15)
    Rectangle (154,5 125x31), "%s", text variable: m_Input_LIGNE_EAU.mnemo
    Frame (76,10 42x40)
        shows VISU_VANNE_2P_H_ACT2(m_Input_VANNE := m_Input_LIGNE_EAU.VEx)
        p1022016623: m_Input_LIGNE_EAU.VEx
    Image (276,1 39x37), invisible if: NOT m_Input_LIGNE_EAU.STATE_NOK, image: MesImages.warning
END_VISUALIZATION

// ---- Visualizations/Symbole/SERVITUDES/VISU_LIGNE_EAU_NO_DEXT.TcVIS
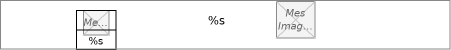
VISUALIZATION VISU_LIGNE_EAU_NO_DEXT  // 451x50
VAR_IN_OUT
	m_Input_LIGNE_EAU : BLOCK_LIGNE_REF;
END_VAR
    Polyline (451,20)
    Polyline (80,20)
    Polyline (129,20)
    Polygon (140,20)
    Polygon (317,20)
    Rectangle (154,5 125x31), "%s", text variable: m_Input_LIGNE_EAU.mnemo
    Frame (76,10 42x40)
        shows VISU_VANNE_2P_H_ACT2(m_Input_VANNE := m_Input_LIGNE_EAU.VEx)
        p1022016623: m_Input_LIGNE_EAU.VEx
    Image (276,1 39x37), invisible if: NOT m_Input_LIGNE_EAU.STATE_NOK, image: MesImages.warning
END_VISUALIZATION

// ---- Visualizations/Symbole/SERVITUDES/VISU_LIGNE_EAU_FLOWTEMP.TcVIS
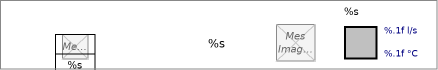
VISUALIZATION VISU_LIGNE_EAU_FLOWTEMP  // 438x70
VAR_IN_OUT
	m_Input_LIGNE_EAU : BLOCK_LIGNE_REF_FLOWTEMP;
END_VAR
    Polyline (451,20)
    Polyline (80,20)
    Polyline (129,20)
    Polygon (140,20)
    Polygon (317,20)
    Rectangle (154,28 125x31), "%s", text variable: m_Input_LIGNE_EAU.mnemo
    Frame (51,30 42x40)
        shows VISU_VANNE_2P_H(m_Input_VANNE := m_Input_LIGNE_EAU.VEx)
        p1022016623: m_Input_LIGNE_EAU.VEx
    Image (276,24 39x37), invisible if: NOT m_Input_LIGNE_EAU.STATE_NOK, image: MesImages.warning
    Rectangle (381,23 45x15), "%.1f l/s", text variable: m_Input_LIGNE_EAU.DEx.STATE_Flow, invisible if: m_Input_LIGNE_EAU.CONF_Max_Flow = 0 AND m_Input_LIGNE_EAU.CONF_Min_Flow = 0
    Rectangle (341,0 36x23), "%s", text variable: m_Input_LIGNE_EAU.mnemo_DEX
    Rectangle (344,26 33x33), colour toggle: m_Input_LIGNE_EAU.STATE_DexT AND m_Input_LIGNE_EAU.VEx.STATE_On
    Polyline (16,8)
    Polyline (24,15)
    Rectangle (381,46 45x15), "%.1f °C", text variable: m_Input_LIGNE_EAU.DEx.STATE_Temp
END_VISUALIZATION

// ---- Visualizations/Symbole/SERVITUDES/VISU_LIGNE_EAU_No_VE.TcVIS
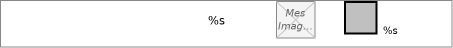
VISUALIZATION VISU_LIGNE_EAU_No_VE  // 453x48
VAR_IN_OUT
	m_Input_LIGNE_EAU : BLOCK_LIGNE_REF;
END_VAR
    Polyline (451,20)
    Polyline (80,20)
    Polyline (129,20)
    Polygon (140,20)
    Polygon (317,20)
    Rectangle (380,15 65x31), "%s", text variable: m_Input_LIGNE_EAU.mnemo_DEX, invisible if: m_Input_LIGNE_EAU.CONF_NO_DexT
    Rectangle (344,1 33x33), colour toggle: (m_Input_LIGNE_EAU.IN_DExT) <> 0, invisible if: (m_Input_LIGNE_EAU.CONF_NO_DexT) <> 0
    Polyline (16,8)
    Polyline (24,15)
    Rectangle (154,5 125x31), "%s", text variable: m_Input_LIGNE_EAU.mnemo
    Image (276,1 39x37), invisible if: NOT m_Input_LIGNE_EAU.STATE_NOK, image: MesImages.warning
END_VISUALIZATION

// ---- Visualizations/Symbole/SERVITUDES/VISU_TEMPRO_PLUS_90.TcVIS
